// TIA Portal project "SimpleHmi" (V13)

(* hardware
DEVICE "S7-1200 station_1"  S7-1200 Station
   slot 0: "Rack_0"  Rack  V1.0
   slot 1: "PLC_1"  CPU 1212C DC/DC/Rly  6ES7 212-1HE40-0XB0  V4.1
*)

// ===== PLC "PLC_1"  CPU 1212C DC/DC/Rly =====

DATA_BLOCK "DB1"   // DB1
{ S7_Optimized_Access := 'FALSE' }
VERSION : 0.1
   VAR
      "Start PB" : Bool;
      "Stop PB" : Bool;
      "Pump Contactor" : Bool;
      "High level limit switch_1" : Bool;
      "Low level limit switch" : Bool;
      "Tank level" : Int;
   END_VAR
BEGIN
END_DATA_BLOCK

DATA_BLOCK "DB2"   // DB2
{ S7_Optimized_Access := 'FALSE' }
VERSION : 0.1
   VAR
      T1 : IEC_TIMER;
      "clock 100ms" : Bool;
   END_VAR
BEGIN
END_DATA_BLOCK

ORGANIZATION_BLOCK "Main"   // OB1, LAD, ProgramCycle
TITLE = "Main Program Sweep (Cycle)"
{ S7_Optimized_Access := 'FALSE' }
VERSION : 0.1
BEGIN

REGION Network 1
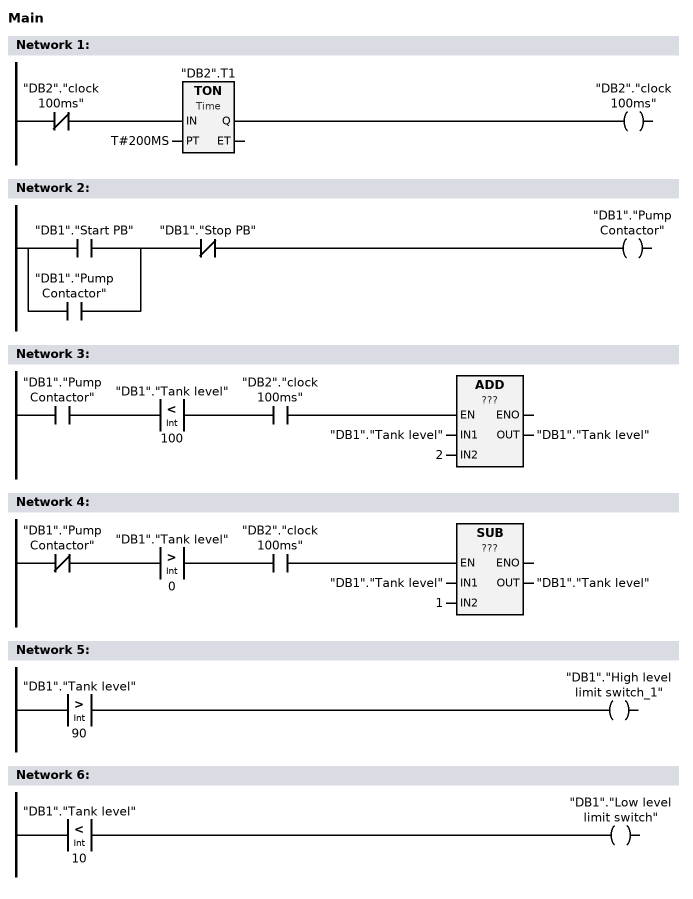
   "DB2".T1.TON(IN := NOT "DB2"."clock 100ms", PT := T#200MS);
   "DB2"."clock 100ms" := "DB2".T1.Q;
END_REGION

REGION Network 2
   RUNG wire#powerrail
      Contact( "DB1"."Start PB" )
      wire#w1
      I_Contact( "DB1"."Stop PB" )
      Coil( "DB1"."Pump Contactor" )
   END_RUNG
   RUNG wire#powerrail
      Contact( "DB1"."Pump Contactor" )
   END_RUNG wire#w1
   // the same network as SCL:
   "DB1"."Pump Contactor" := ("DB1"."Start PB" OR "DB1"."Pump Contactor") AND NOT "DB1"."Stop PB";
END_REGION

REGION Network 3
   RUNG wire#powerrail
      Contact( "DB1"."Pump Contactor" )
      { S7_Templates := "SrcType := Int" } LT_Contact(in1 := "DB1"."Tank level", in2 := 100)
      Contact( "DB2"."clock 100ms" )
      { S7_Templates := "SrcType := ???" } Add(in1 := "DB1"."Tank level", in2 := 2, out => "DB1"."Tank level")
   END_RUNG
   // the same network as SCL:
   IF "DB1"."Pump Contactor" AND ("DB1"."Tank level" < 100) AND "DB2"."clock 100ms" THEN
       "DB1"."Tank level" := "DB1"."Tank level" + 2;
   END_IF;
END_REGION

REGION Network 4
   RUNG wire#powerrail
      I_Contact( "DB1"."Pump Contactor" )
      { S7_Templates := "SrcType := Int" } GT_Contact(in1 := "DB1"."Tank level", in2 := 0)
      Contact( "DB2"."clock 100ms" )
      { S7_Templates := "SrcType := ???" } Sub(in1 := "DB1"."Tank level", in2 := 1, out => "DB1"."Tank level")
   END_RUNG
   // the same network as SCL:
   IF NOT "DB1"."Pump Contactor" AND ("DB1"."Tank level" > 0) AND "DB2"."clock 100ms" THEN
       "DB1"."Tank level" := "DB1"."Tank level" - 1;
   END_IF;
END_REGION

REGION Network 5
   RUNG wire#powerrail
      { S7_Templates := "SrcType := Int" } GT_Contact(in1 := "DB1"."Tank level", in2 := 90)
      Coil( "DB1"."High level limit switch_1" )
   END_RUNG
   // the same network as SCL:
   "DB1"."High level limit switch_1" := "DB1"."Tank level" > 90;
END_REGION

REGION Network 6
   RUNG wire#powerrail
      { S7_Templates := "SrcType := Int" } LT_Contact(in1 := "DB1"."Tank level", in2 := 10)
      Coil( "DB1"."Low level limit switch" )
   END_RUNG
   // the same network as SCL:
   "DB1"."Low level limit switch" := "DB1"."Tank level" < 10;
END_REGION
END_ORGANIZATION_BLOCK